Staubli VAL3: F5_start.pgx

public program F5_start()
begin
  //start Synchronous move
  if bTxtPrSv==false
    //    popUpMsg("请首先对点位文件初始化（按F3-PoIn）")
    TcpStrRec:nFeedback=532
  else

    socket="(RBSTAT)"
    delay(0.01)
    nTime=0
    nTestNum=0
    if taskStatus("SychMove")==-1
      taskCreateSync "SychMove",0.004,bRes,sychronMove()
      //taskCreateSync "SychMove",0.008,bRes,sychronRealM()
    else
      popUpMsg("Task is already running")
    endIf
  endIf
  //call sychronMove()
end
